# EPICS autosave request: utcaApp/Db/rtmlamp_channel.req
$(S)$(RTM_CHAN)CurrLoopKp-SP
$(S)$(RTM_CHAN)CurrLoopTi-SP
$(S)$(RTM_CHAN)CurrGain-SP
$(S)$(RTM_CHAN)CurrOffset-SP
$(S)$(RTM_CHAN)VoltGain-SP
$(S)$(RTM_CHAN)VoltOffset-SP
$(S)$(RTM_CHAN)Current-SP
$(S)$(RTM_CHAN)Voltage-SP
$(S)$(RTM_CHAN)TrigEn-Sel
